PROGRAM MAIN
VAR
END_VAR

Process();

END_PROGRAM

(* stored: Version 1.1.0.1, ProductVersion 3.1.4022.12
   POU MAIN: Id {9f23c54e-5031-461b-a33a-312d95aabe56}, SpecialFunc None *)
